// TwinCAT 3 PLC project QuadratureEncoder
// ProgramVersion: 3.1.4024.0
// libraries:
//   Tc2_Standard, * (Beckhoff Automation GmbH)
//   Tc2_System, * (Beckhoff Automation GmbH)
//   Tc3_Module, * (Beckhoff Automation GmbH)
// project tree:
//   GVLs/ GVL.TcGVL
//   / PlcTask.TcTTO
//   POUs/ MAIN.TcPOU, FB_QuadratureEncoder.TcPOU (not stored)
// real-time tasks:
//   TASK PlcTask: cycle T#10ms, priority 20, ADS port 350
// I/O:
//   DEVICE Device 2 (EtherCAT), AmsNetId 141.212.76.55.3.1
//     Term 1 (EK1100) [EK1100 EtherCAT Coupler (2A E-Bus)]
//       Term 2 (EL4038) [EL4038 8Ch. Ana. Output +/-10V, 12bit]
//       Term 3 (EL3174) [EL3174 4Ch. Ana. Input +/-10V Diff., +/-20mA SingleEnded, 16 Bit]
//       Term 4 (EL5122) [EL5122 2Ch. Inc. Encoder 5V (2xAB TTL)]
//       Term 5 (EL9011) [EL9011 End Terminal]
// variable links:
//   QuadratureEncoder/QuadratureEncoder Instance <-> Device 2 (EtherCAT)/Term 1 (EK1100)/Term 4 (EL5122)
//     PlcTask Inputs/MAIN.QuadratureEncoder_C1.QE_CHANNEL.MDP5001_511_Input/MDP5001_511_Counter_value <-> ENC Status Channel 1/Counter value
//     PlcTask Inputs/MAIN.QuadratureEncoder_C1.QE_CHANNEL.MDP5001_511_Input/MDP5001_511_Latch_value <-> ENC Status Channel 1/Latch value
//     PlcTask Inputs/MAIN.QuadratureEncoder_C1.QE_CHANNEL.MDP5001_511_Input/MDP5001_511_Status <-> ENC Status Channel 1/Status
//     PlcTask Outputs/MAIN.QuadratureEncoder_C1.QE_CHANNEL.MDP5001_511_Output/MDP5001_511_Control <-> ENC Control Channel 1/Control
//     PlcTask Outputs/MAIN.QuadratureEncoder_C1.QE_CHANNEL.MDP5001_511_Output/MDP5001_511_Set_counter_value <-> ENC Control Channel 1/Set counter value

CONFIGURATION QuadratureEncoder
    RESOURCE PLC ON TwinCAT3
        TASK PlcTask(INTERVAL := T#10ms, PRIORITY := 20);
        PROGRAM MAIN WITH PlcTask : MAIN;
    END_RESOURCE
END_CONFIGURATION

// ---- GVLs/GVL.TcGVL
{attribute 'qualified_only'}
VAR_GLOBAL
	Encoder1NetCounts : LINT; 
	Encoder1Degrees : REAL; 
END_VAR

// ---- POUs/MAIN.TcPOU
PROGRAM MAIN
VAR
	QuadratureEncoder_C1 : FB_QuadratureEncoder; 
END_VAR

// Update encoder reading 
QuadratureEncoder_C1(); // This internally calls everything else we need
GVL.Encoder1NetCounts := QuadratureEncoder_C1.nNetCounts; 
GVL.Encoder1Degrees := QuadratureEncoder_C1.rDegrees;

END_PROGRAM
